% RSLogix 500 project P6_HOURMETER.RSS, saved by version 8.30.00.16 %
PROJECT "P6"    % processor: Bul.1763 MicroLogix 1100 Series B %

PROGRAM FILES
  LAD 2   6 rungs

DATA FILES
  O0 OUTPUT  4 elements
  I1 INPUT  6 elements
  S2 STATUS  66 elements
  B3 BINARY  1 elements
  T4 TIMER  1 elements
  C5 COUNTER  5 elements
  R6 CONTROL  1 elements
  N7 INTEGER  15 elements
  F8 FLOAT  1 elements

LADDER 2
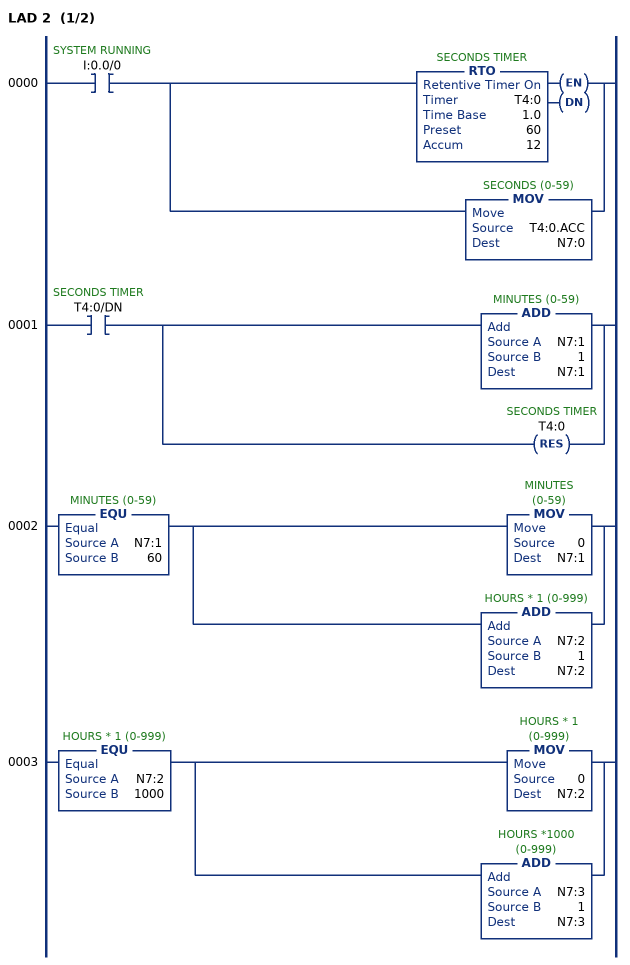
% Rung: 0 %
SOR XIC I:0.0/0 BST RTO T4:0 1.0 60 12 NXB MOV T4:0.ACC N7:0 BND EOR
%   I:0.0/0  "SYSTEM RUNNING" %
%   T4:0  "SECONDS TIMER" %
%   N7:0  "SECONDS (0-59)" %
% Rung: 1 %
SOR XIC T4:0/DN BST ADD N7:1 1 N7:1 NXB RES T4:0 BND EOR
%   T4:0  "SECONDS TIMER" %
%   N7:1  "MINUTES (0-59)" %
% Rung: 2 %
SOR EQU N7:1 60 BST MOV 0 N7:1 NXB ADD N7:2 1 N7:2 BND EOR
%   N7:1  "MINUTES (0-59)" %
%   N7:2  "HOURS * 1 (0-999)" %
% Rung: 3 %
SOR EQU N7:2 1000 BST MOV 0 N7:2 NXB ADD N7:3 1 N7:3 BND EOR
%   N7:2  "HOURS * 1 (0-999)" %
%   N7:3  "HOURS *1000 (0-999)" %

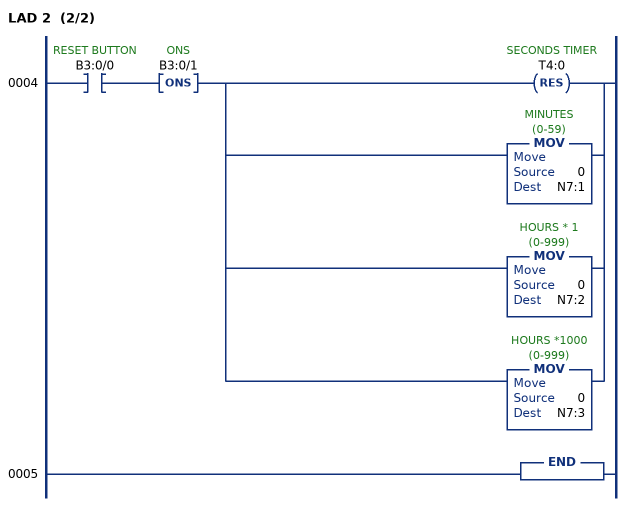
% Rung: 4 %
SOR XIC B3:0/0 ONS B3:0/1 BST RES T4:0 NXB MOV 0 N7:1 NXB MOV 0 N7:2 NXB MOV 0 N7:3 BND EOR
%   B3:0/0  "RESET BUTTON" %
%   B3:0/1  "ONS" %
%   T4:0  "SECONDS TIMER" %
%   N7:1  "MINUTES (0-59)" %
%   N7:2  "HOURS * 1 (0-999)" %
%   N7:3  "HOURS *1000 (0-999)" %
% Rung: 5 %
SOR END EOR

OTHER DOCUMENTED ADDRESSES
  C5:0  "MINUTES COUNTER"
  C5:1  "HOURS*1 COUNTER"
  C5:2  "HOURS COUNTER*1000"
  C5:3  "HOURS COUNTER *1000 (0-999)"

DATA TABLE (non-zero values as saved)
DATA T4
% .PRE .ACC %
% T4:0 % 60 12
DATA C5
% .PRE .ACC %
% C5:0 % 60 60
% C5:1 % 999 1
% C5:2 % 999 0
DATA N7
% N7:0 % 12 2 0 1000 0 0 0 0 0 0
